FUNCTION_BLOCK FileLogger IMPLEMENTS EventLogger
VAR_INPUT
END_VAR
VAR_OUTPUT
  error_id: DWORD;
END_VAR
VAR
  _path: STRING(255);
  file: TcExt.FileMemory;
  localtime: FB_LocalSystemTime := (bEnable:=TRUE);
  _done: BOOL;
  _level: EventLevel;
END_VAR

PROPERTY done : BOOL
GET
done := _done;
END_GET
SET // PRIVATE
_done := done;
END_SET
END_PROPERTY

METHOD PRIVATE get_timestaped_path : STRING(255)
VAR
  datetime: STRING(255);
  char_at: INT;
END_VAR
datetime := SYSTEMTIME_TO_STRING(localtime.systemTime);

char_at := FIND(datetime, '.');
IF char_at <> 0 THEN
  datetime := DELETE(datetime, 4, char_at);
END_IF

REPEAT
  char_at := FIND(datetime, ':');
  IF char_at <> 0 THEN
    datetime := REPLACE(datetime, '_', 1, char_at);
  END_IF
UNTIL char_at = 0
END_REPEAT

get_timestaped_path := CONCAT(path, CONCAT('log_', CONCAT(datetime, '.log')));
END_METHOD

PROPERTY PUBLIC level : EventLevel
GET
level := _level;
END_GET
SET
_level := level;
END_SET
END_PROPERTY

PROPERTY path : STRING(255)
GET
path := _path;
END_GET
SET
_path := path;
END_SET
END_PROPERTY

METHOD save
VAR_INPUT
  execute: BOOL;
  data_ptr: PVOID;
  data_size: DWORD;
END_VAR
VAR_INST
  r_execute: R_TRIG;
END_VAR
localtime();
r_execute(CLK:=execute);

IF r_execute.Q THEN
  file.path := get_timestaped_path();
END_IF
file.write(
  start:=execute,
  data_ptr:=data_ptr,
  data_size:=data_size,
  done=>_done,
  error_id=>error_id);
END_METHOD

METHOD submit_event_message
VAR_INPUT
	ev: EventMessage;
END_VAR
END_METHOD

END_FUNCTION_BLOCK

(* stored: Version 1.1.0.1, ProductVersion 3.1.4024.9
   POU FileLogger: Id {eddd5bf2-9f8b-4014-b1a1-2b9514f6af17}, SpecialFunc None
   Property done: Id {687b28e8-dfd4-40db-a439-a623577f86e7}
   Get Get: Id {f4b573f4-12a0-4d9f-ade5-ca186ec28527}
   Set Set: Id {79f34a29-2418-4485-9442-9987efedfe83}
   Method get_timestaped_path: Id {fd365ee7-137c-43d5-b097-a6c91d56c64b}
   Property level: Id {ab6b9969-76e1-4879-b617-99481726f092}
   Get Get: Id {5ab1af13-9930-49f3-9811-710132aa1fb1}
   Set Set: Id {cf7d265b-a08f-46d3-959d-33b6de9e6222}
   Property path: Id {8ad77a76-a7ae-4211-a029-62cbfb7f3a1a}
   Get Get: Id {32fab473-3ae0-4d2e-b9ac-c6915164202f}
   Set Set: Id {b4db1cae-d219-49b1-923d-846a377b7031}
   Method save: Id {501c7d54-f5c2-48f2-862f-f63db1339f45}
   Method submit_event_message: Id {4532367b-994f-48dd-829f-58c767e7db29} *)
